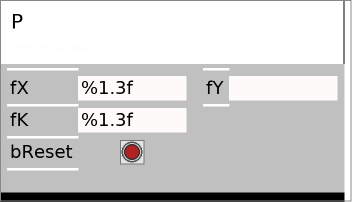
VISUALIZATION RET_VISU_P  // 352x202
VAR_INPUT
   {attribute 'parameterstringof' := 'm_Input_FB'}
   m_Input_INST_Str : STRING;
END_VAR
VAR_IN_OUT
   m_Input_FB : P;
END_VAR
    RoundedRectangle (0,0 344x81)
    RoundedRectangle (0,162 344x40)
    Rectangle (0,64 344x128)
    PushSwitch (120,140 24x24), variable: m_Input_FB.bReset, behaviour: TOGGLE, style: Switch-PushSwitch-Red
    Rectangle (8,8 344x27), "P"
    Rectangle (8,35 344x27), "Instance: %s", text variable: m_Input_INST_Str
    Rectangle (7,68 71x2)
    Rectangle (78,76 108x24), "%1.3f", text variable: m_Input_FB.fX
        OnMouseClick: write the text variable via Default
    Rectangle (7,76 71x24), "fX"
    Rectangle (7,104 71x2)
    Rectangle (78,108 108x24), "%1.3f", text variable: m_Input_FB.fK
        OnMouseClick: write the text variable via Default
    Rectangle (7,108 71x24), "fK"
    Rectangle (7,136 71x2)
    Rectangle (7,140 71x24), "bReset"
    Rectangle (7,168 71x2)
    Rectangle (203,68 26x2)
    Rectangle (229,76 108x24), text variable: m_Input_FB.fY
    Rectangle (203,76 26x24), "fY"
    Rectangle (203,104 26x2)
END_VISUALIZATION

(* stored: Version 1.1.0.1, ProductVersion 3.1.4024.12
   Visu RET_VISU_P: Id {90fae039-4467-4794-9906-0c71927510f0} *)
